
FUNCTION CB_dint_to_bool : BOOL


TITLE = ' Convert a double integer into an boolean '
VERSION : '1.0'
AUTHOR  : CB
NAME    : DintToBo
FAMILY  : TNI

VAR_INPUT
    IN : DINT;
END_VAR

VAR_TEMP

END_VAR

BEGIN

CB_dint_to_bool := DINT_TO_BOOL(IN);

END_FUNCTION
